FUNCTION_BLOCK FB_RPC
VAR_INPUT
END_VAR
VAR_OUTPUT
END_VAR
VAR
	m_cnt_add : UINT;
END_VAR

{attribute 'TcRpcEnable'}
METHOD M_Add : DINT
VAR_INPUT
	a : DINT;
	b : DINT;
END_VAR
m_cnt_add := m_cnt_add +1;
M_Add := a + b;
END_METHOD

END_FUNCTION_BLOCK

(* stored: Version 1.1.0.1, ProductVersion 3.1.4024.12
   POU FB_RPC: Id {af2183e0-0c72-4425-8a40-087ae260afdf}, SpecialFunc None
   Method M_Add: Id {dc8a013e-80a7-4de8-a7fa-97726564522d} *)
